INTERFACE I_TankController

METHOD ApplyCooling
VAR_IN_OUT	
	refTank : ST_Tank;
END_VAR
END_METHOD

METHOD CheckSafety : BOOL
VAR_INPUT
	pTank : POINTER TO ST_Tank;
END_VAR

VAR_OUTPUT
	alarm : BOOL;
END_VAR
END_METHOD

END_INTERFACE

(* stored: Version 1.1.0.1, ProductVersion 3.1.4024.16
   Itf I_TankController: Id {7c40f9a2-9de0-4c10-aa60-c6e7596dc1c3}
   Method ApplyCooling: Id {bd3ade69-d84b-4eff-a3f9-a660017a672e}
   Method CheckSafety: Id {9418bb1b-fde8-466b-aa58-e222770778d9} *)
